(* Schneider Machine Expert - Basic project 1, file version 1.7.0.0 *)
(* ProjectInformations: Name=New project *)

HARDWARE
  Cpu 0: TM221M16R/G
  EthernetConfiguration: NetworkName=M221, IpAllocationMode=FixedAddress, IpAddress=0.0.0.0, SubnetMask=0.0.0.0
  SerialLineConfiguration: Baud=Baud19200, Parity=ParityEven, DataBits=DataBits8, StopBits=StopBits1, PhysicalMedium=PhysicalMediumRs485, TransmissionMode=TransmissionModeModbusRtu, SlaveId=1, Addressing=SlaveAddressing
  MastTask: UsePeriodScanMode=false, PeriodScan=100
  FastTask: Period=255
  CpuBehavior: StartingMode=StartAsPreviousState, AutoSaveRamOnEeprom=true, WatchdogPeriod=250

SYMBOLS  (address, symbol, comment, settings)
  %IW0.0      [Type=Type_0_10V, Scope=Scope_Normal, Minimum=0, Maximum=1000]

POU New POU
  (* SectionNumber=1 *)

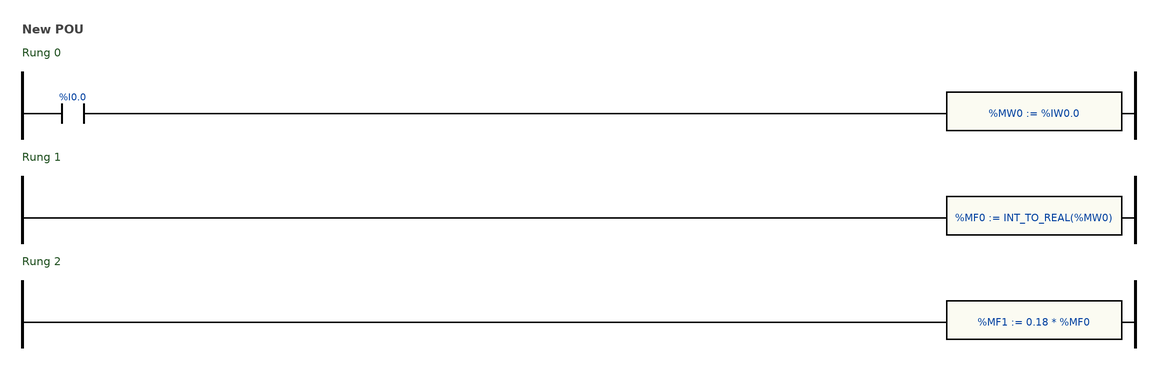

// Rung 0
  LD %I0.0
  [ %MW0 := %IW0.0 ]
  // as ST:
  //   IF %I0.0 THEN %MW0 := %IW0.0; END_IF;

// Rung 1
  LD 1
  [ %MF0 := INT_TO_REAL ( %MW0 ) ]
  // as ST:
  //   %MF0 := INT_TO_REAL ( %MW0 );

// Rung 2
  LD 1
  [ %MF1 := 0.18 * %MF0 ]
  // as ST:
  //   %MF1 := 0.18  *  %MF0;
